TYPE PiperCommand :
STRUCT
	Abort : BOOL;
	Start : BOOL;
	Stop : BOOL;
	Clear : BOOL;
	Reset : BOOL;
	Suspend : BOOL;
	Unsuspend : BOOL;
	Hold : BOOL;
	Unhold : BOOL;
END_STRUCT
END_TYPE;

(* stored: Version 1.1.0.1, ProductVersion 3.1.4024.12
   DUT PiperCommand: Id {a07f4fb2-d61e-4e2a-9ec5-433dc322d33c} *)
